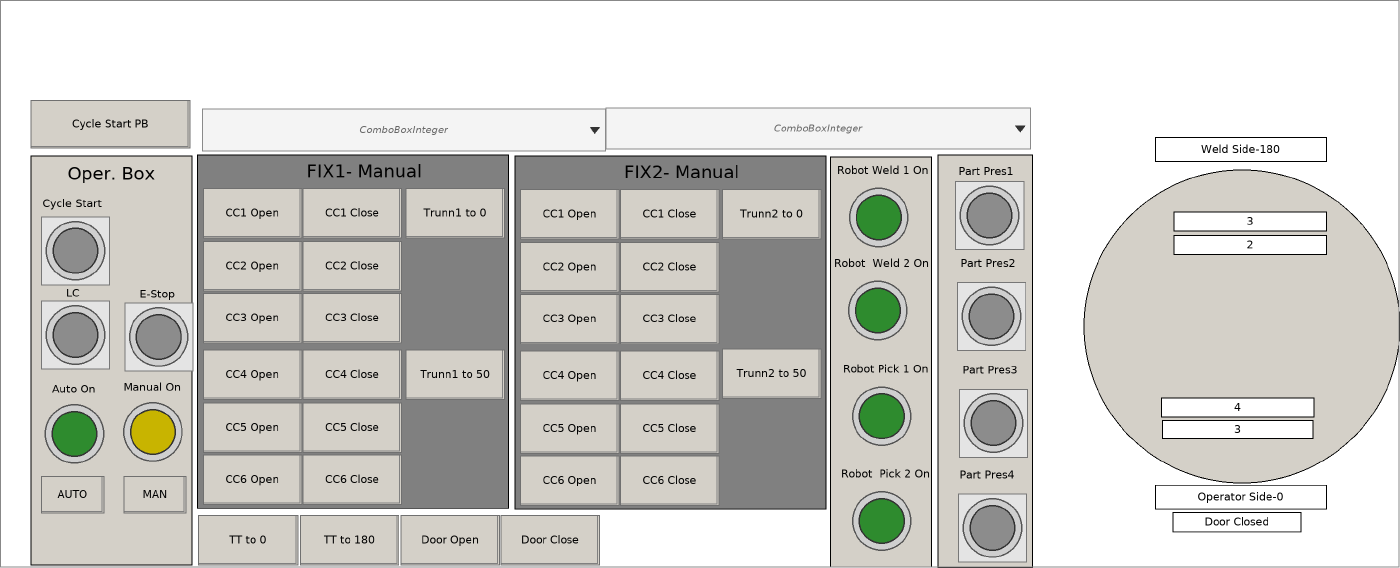
VISUALIZATION Visualization  // 1429x580
    Rectangle (957,158 97x422)
    Rectangle (847,160 104x419)
    Rectangle (31,159 165x418)
    PushSwitchLed (973,185 74x70), variable: MAIN.PartPresent1, behaviour: TOGGLE, style: Switch-PushSwitchLed-Gray
    Label (964,160 89x30), "Part Pres1"
    PushSwitchLed (40,221 74x70), variable: MAIN.CycleStart, behaviour: TOGGLE, style: Switch-PushSwitchLed-Gray
    Label (29,193 90x30), "Cycle Start"
    PushSwitchLed (975,288 74x70), variable: MAIN.PartPresent2, behaviour: TOGGLE, style: Switch-PushSwitchLed-Gray
    Label (964,254 89x30), "Part Pres2"
    Button (42,486 64x38), "AUTO", text variable: MAIN.HMI_Auto, colour toggle: MAIN.HMI_Auto
        tap MAIN.HMI_Auto
    PushSwitchLed (977,397 74x70), variable: MAIN.PartPresent3, behaviour: TOGGLE, style: Switch-PushSwitchLed-Gray
    PushSwitchLed (976,504 74x70), variable: MAIN.PartPresent4, behaviour: TOGGLE, style: Switch-PushSwitchLed-Gray
    Label (965,470 89x30), "Part Pres4"
    Label (966,363 89x30), "Part Pres3"
    PushSwitchLed (125,309 74x70), variable: MAIN.EmergencyStop, behaviour: TOGGLE, style: Switch-PushSwitchLed-Gray
    Label (116,288 89x25), "E-Stop"
    Label (30,287 89x25), "LC"
    PushSwitchLed (40,307 74x70), variable: MAIN.LightCurtainOK, behaviour: TOGGLE, style: Switch-PushSwitchLed-Gray
    Lamp1 (862,187 70x70), variable: MAIN.Robot1.Weld1Active, style: Lamp-Lamp1-Green
    Label (850,159 102x30), "Robot Weld 1 On"
    Lamp1 (861,282 70x70), variable: MAIN.Robot1.Weld2Active, style: Lamp-Lamp1-Green
    Label (849,254 102x30), "Robot Weld 2 On"
    Lamp1 (41,408 70x70), variable: MAIN.ModeMgr.AutoMode, style: Lamp-Lamp1-Green
    Label (31,385 89x25), "Auto On"
    Button (126,486 64x38), "MAN", text variable: MAIN.HMI_Manual, colour toggle: MAIN.HMI_Manual
        tap MAIN.HMI_Manual
    ComboBoxInteger (206,111 412x43), variable: MAIN.AutoSeq.State1, text list: 'TextList_State1'
    ComboBoxInteger (618,110 434x42), variable: MAIN.AutoSeq.State2, text list: 'TextList_State2'
    Lamp1 (121,406 70x70), variable: MAIN.ModeMgr.ManualMode, style: Lamp-Lamp1-Yellow
    Label (111,383 89x25), "Manual On"
    Label (8,166 211x23), "Oper. Box"
    Ellipse (1106,173 323x320)
    Rectangle (1186,429 154x19), "1", colour toggle: MAIN.Trunnion1.At0, invisible if: MAIN.Turntable.At180
    Rectangle (1185,406 156x20), "2", colour toggle: MAIN.Trunnion1.At50, invisible if: MAIN.Turntable.At180
    Rectangle (1186,429 154x19), "3", colour toggle: MAIN.Trunnion2.At0, invisible if: MAIN.Turntable.At0
    Rectangle (1185,406 156x20), "4", colour toggle: MAIN.Trunnion2.At50, invisible if: MAIN.Turntable.At0
    Rectangle (1198,240 156x20), "4", colour toggle: MAIN.Trunnion2.At50, invisible if: MAIN.Turntable.At180
    Rectangle (1198,216 156x20), "1", colour toggle: MAIN.Trunnion1.At0, invisible if: MAIN.Turntable.At0
    Rectangle (1198,240 156x20), "2", colour toggle: MAIN.Trunnion1.At50, invisible if: MAIN.Turntable.At0
    Rectangle (1198,216 156x20), "3", colour toggle: MAIN.Trunnion2.At0, invisible if: MAIN.Turntable.At180
    Rectangle (1179,140 175x25), "Weld Side-180", colour toggle: MAIN.Turntable.At180
    Rectangle (1179,495 175x25), "Operator Side-0", colour toggle: MAIN.Turntable.At0
    Rectangle (1197,523 131x20), "Door Opened", colour toggle: MAIN.RollerDoor1.OpenedSim, invisible if: MAIN.RollerDoor1.ClosedSim
    Rectangle (1197,523 131x20), "Door Closed", colour toggle: MAIN.RollerDoor1.ClosedSim, invisible if: MAIN.RollerDoor1.OpenedSim
    Button (31,102 163x49), "Cycle Start PB", text variable: MAIN.CycleStart, colour toggle: MAIN.CycleStart
        tap MAIN.CycleStart
    Rectangle (201,158 318x361)
    Button (202,526 102x51), "TT to 0", text variable: MAIN.Turntable.At0, colour toggle: MAIN.Turntable.At0
        tap MAIN.ManTT0
    Button (306,526 101x51), "TT to 180", text variable: MAIN.Turntable.At180, colour toggle: MAIN.Turntable.At180
        tap MAIN.ManTT180
    Button (414,192 101x51), "Trunn1 to 0", text variable: MAIN.Trunnion1.At0, colour toggle: MAIN.Trunnion1.At0
        tap MAIN.ManTrn10
    Button (414,357 101x51), "Trunn1 to 50", text variable: MAIN.Trunnion1.At50, colour toggle: MAIN.Trunnion1.At50
        tap MAIN.ManTrn150
    Button (309,192 101x51), "CC1 Close", text variable: MAIN.Fixture_1_CC1.ClosedSim, colour toggle: MAIN.Fixture_1_CC1.ClosedSim
        tap MAIN.Fixture_1_ManCC1Close
    Button (207,192 101x51), "CC1 Open", text variable: MAIN.Fixture_1_CC1.OpenedSim, colour toggle: MAIN.Fixture_1_CC1.OpenedSim
        tap MAIN.Fixture_1_ManCC1Open
    Label (242,155 260x40), "FIX1- Manual"
    Button (409,526 101x51), "Door Open", text variable: MAIN.RollerDoor1.OpenedSim, colour toggle: MAIN.RollerDoor1.OpenedSim
        tap MAIN.ManRollerDoor1Open
    Button (511,526 101x51), "Door Close", text variable: MAIN.RollerDoor1.ClosedSim, colour toggle: MAIN.RollerDoor1.ClosedSim
        tap MAIN.ManRollerDoor1Close
    Lamp1 (865,390 70x70), variable: MAIN.Robot2.Pick1Active, style: Lamp-Lamp1-Green
    Label (853,362 102x30), "Robot Pick 1 On"
    Lamp1 (865,497 70x70), variable: MAIN.Robot2.Pick2Active, style: Lamp-Lamp1-Green
    Label (853,469 102x30), "Robot Pick 2 On"
    Button (309,246 101x51), "CC2 Close", text variable: MAIN.Fixture_1_CC2.ClosedSim, colour toggle: MAIN.Fixture_1_CC2.ClosedSim
        tap MAIN.Fixture_1_ManCC2Close
    Button (207,246 101x51), "CC2 Open", text variable: MAIN.Fixture_1_CC2.OpenedSim, colour toggle: MAIN.Fixture_1_CC2.OpenedSim
        tap MAIN.Fixture_1_ManCC2Open
    Button (207,299 101x51), "CC3 Open", text variable: MAIN.Fixture_1_CC3.OpenedSim, colour toggle: MAIN.Fixture_1_CC3.OpenedSim
        tap MAIN.Fixture_1_ManCC3Open
    Button (309,299 101x51), "CC3 Close", text variable: MAIN.Fixture_1_CC3.ClosedSim, colour toggle: MAIN.Fixture_1_CC3.ClosedSim
        tap MAIN.Fixture_1_ManCC3Close
    Button (207,357 101x51), "CC4 Open", text variable: MAIN.Fixture_1_CC4.OpenedSim, colour toggle: MAIN.Fixture_1_CC4.OpenedSim
        tap MAIN.Fixture_1_ManCC4Open
    Button (309,357 101x51), "CC4 Close", text variable: MAIN.Fixture_1_CC4.ClosedSim, colour toggle: MAIN.Fixture_1_CC4.ClosedSim
        tap MAIN.Fixture_1_ManCC4Close
    Button (309,411 101x51), "CC5 Close", text variable: MAIN.Fixture_1_CC5.ClosedSim, colour toggle: MAIN.Fixture_1_CC5.ClosedSim
        tap MAIN.Fixture_1_ManCC5Close
    Button (207,411 101x51), "CC5 Open", text variable: MAIN.Fixture_1_CC5.OpenedSim, colour toggle: MAIN.Fixture_1_CC5.OpenedSim
        tap MAIN.Fixture_1_ManCC5Open
    Button (207,464 101x51), "CC6 Open", text variable: MAIN.Fixture_1_CC6.OpenedSim, colour toggle: MAIN.Fixture_1_CC6.OpenedSim
        tap MAIN.Fixture_1_ManCC6Open
    Button (309,464 101x51), "CC6 Close", text variable: MAIN.Fixture_1_CC6.ClosedSim, colour toggle: MAIN.Fixture_1_CC6.ClosedSim
        tap MAIN.Fixture_1_ManCC6Close
    Rectangle (525,159 318x361)
    Button (633,193 101x51), "CC1 Close", text variable: MAIN.Fixture_2_CC1.ClosedSim, colour toggle: MAIN.Fixture_2_CC1.ClosedSim
        tap MAIN.Fixture_2_ManCC1Close
    Button (531,193 101x51), "CC1 Open", text variable: MAIN.Fixture_2_CC1.OpenedSim, colour toggle: MAIN.Fixture_2_CC1.OpenedSim
        tap MAIN.Fixture_2_ManCC1Open
    Label (566,156 260x40), "FIX2- Manual"
    Button (633,247 101x51), "CC2 Close", text variable: MAIN.Fixture_2_CC2.ClosedSim, colour toggle: MAIN.Fixture_2_CC2.ClosedSim
        tap MAIN.Fixture_2_ManCC2Close
    Button (531,247 101x51), "CC2 Open", text variable: MAIN.Fixture_2_CC2.OpenedSim, colour toggle: MAIN.Fixture_2_CC2.OpenedSim
        tap MAIN.Fixture_2_ManCC2Open
    Button (531,300 101x51), "CC3 Open", text variable: MAIN.Fixture_2_CC3.OpenedSim, colour toggle: MAIN.Fixture_2_CC3.OpenedSim
        tap MAIN.Fixture_2_ManCC3Open
    Button (633,300 101x51), "CC3 Close", text variable: MAIN.Fixture_2_CC3.ClosedSim, colour toggle: MAIN.Fixture_2_CC3.ClosedSim
        tap MAIN.Fixture_2_ManCC3Close
    Button (531,358 101x51), "CC4 Open", text variable: MAIN.Fixture_2_CC4.OpenedSim, colour toggle: MAIN.Fixture_2_CC4.OpenedSim
        tap MAIN.Fixture_2_ManCC4Open
    Button (633,358 101x51), "CC4 Close", text variable: MAIN.Fixture_2_CC4.ClosedSim, colour toggle: MAIN.Fixture_2_CC4.ClosedSim
        tap MAIN.Fixture_2_ManCC4Close
    Button (633,412 101x51), "CC5 Close", text variable: MAIN.Fixture_2_CC5.ClosedSim, colour toggle: MAIN.Fixture_2_CC5.ClosedSim
        tap MAIN.Fixture_2_ManCC5Close
    Button (531,412 101x51), "CC5 Open", text variable: MAIN.Fixture_2_CC5.OpenedSim, colour toggle: MAIN.Fixture_2_CC5.OpenedSim
        tap MAIN.Fixture_2_ManCC5Open
    Button (531,465 101x51), "CC6 Open", text variable: MAIN.Fixture_2_CC6.OpenedSim, colour toggle: MAIN.Fixture_2_CC6.OpenedSim
        tap MAIN.Fixture_2_ManCC6Open
    Button (633,465 101x51), "CC6 Close", text variable: MAIN.Fixture_2_CC6.ClosedSim, colour toggle: MAIN.Fixture_2_CC6.ClosedSim
        tap MAIN.Fixture_2_ManCC6Close
    Button (737,193 101x51), "Trunn2 to 0", text variable: MAIN.Trunnion2.At0, colour toggle: MAIN.Trunnion2.At0
        tap MAIN.ManTrn20
    Button (737,356 101x51), "Trunn2 to 50", text variable: MAIN.Trunnion2.At50, colour toggle: MAIN.Trunnion2.At50
        tap MAIN.ManTrn250
END_VISUALIZATION

(* stored: Version 1.1.0.1, ProductVersion 3.1.4024.16
   Visu Visualization: Id {4a9894a2-80b5-4c53-88d8-0357fa8aba4f} *)
